Staubli VAL3: setCheckRow.pgx

public program setCheckRow(bool x_bCheckUpLim (dimensions=1))
begin
  //-----------------------------------------------------------------------
  //Header begin
  //Description of program
  // This routines activates of de-activates the row number checking parameter
  // This parameter determines wether or not the row number will be checked against
  // the upper limit (400). The check against the lower limit (0) always remains active.
  //
  // Input Parameters
  //  x_bCheckUpLim :
  //    role : set to true to check row number against upper limit of 400 or to false otherwise
  //
  //Examples
  //  call setCheckRow(true)
  //
  //History
  //  Creation : 03-05-11 - CROC
  //Header end
  //-----------------------------------------------------------------------
  bCheckRowUpLim=x_bCheckUpLim
end
